{attribute 'qualified_only'}
{attribute 'strict'}
TYPE CounterState :
(
	STOP, MEASURE, WAIT
);
END_TYPE

(* stored: Version 1.1.0.1, ProductVersion 3.1.4024.12
   DUT CounterState: Id {296f8b49-6762-4f39-87e0-0ca8da1c2a08} *)
